// TIA Portal V17 export
// export: Created 2021-12-03T08:13:05.7304339Z, ExportSetting WithDefaults, DisplayName Totally Integrated Automation Portal, DisplayVersion V17, DisplayName TIA Portal Openness, DisplayVersion V17, DisplayName TIA Portal Version Control Interface, DisplayVersion V17, DisplayName STEP 7 Professional, DisplayVersion V17, DisplayName STEP 7 Safety, DisplayVersion V17, DisplayName WinCC Advanced, DisplayVersion V17
DATA_BLOCK "GDB_SpdClclt"   // DB502
VERSION : 0.1
// stored: AutoNumber false, IsOnlyStoredInLoadMemory false, IsWriteProtectedInAS false
   VAR
      Transit : Struct
         Strt : Bool;   // Старт
         HP : Bool;   // Конвейер в домашней позиции
         TmrStrt : Bool;   // За
         CalcCompl : Bool;
         SeqCompl : Bool;
      END_STRUCT;
      Action : Struct
         Init : Bool;   // Инициализация
         Homming : Bool;   // Возврат в HP
         BwdStrt : Bool;   // Старт
         TmrStrt : Bool;   // Запуск таймера
         Completed : Bool;   // Расчет выполнен
      END_STRUCT;
      SR : Struct
         Run : Bool;
         TmrStrt : Bool;
      END_STRUCT;
      TRIG : Struct
         P_XrayFwd : Bool;
         P_XrayBwd : Bool;
      END_STRUCT;
      Run : Bool;   // Запуск подсчета скорости
      SpdClcltSpNr : Int;   // Номер шага
      RdySpdClclt : Bool;   // Готовность к запуску полсчета скорости
      FactSpeed : Int;   // Фактическая скорость
   END_VAR
BEGIN
END_DATA_BLOCK
